// TwinCAT 3 PLC project Untitled1
// ProgramVersion: 3.1.4024.0
// libraries:
//   Tc2_MC2, * (Beckhoff Automation GmbH)
//   Tc2_NCI, * (Beckhoff Automation GmbH)
//   Tc2_Standard, * (Beckhoff Automation GmbH)
//   Tc2_System, * (Beckhoff Automation GmbH)
//   Tc3_Module, * (Beckhoff Automation GmbH)
//   VisuDialogs, * (System)
//   VisuSymbols,3.5.10.0,System
// project tree:
//   DUTs/ MC_CMD.TcDUT, MC_Status.TcDUT
//   / GlobalTextList.TcGTLO, PlcTask.TcTTO, Visualization Manager.TcVMO (not stored)
//   GVLs/ GVL.TcGVL
//   POUs/ MAIN.TcPOU, PANEL.TcPOU, FB_NCI.TcPOU, FB_PowerAll.TcPOU, X_Axis.TcPOU, Y_Axis.TcPOU, Z_Axis.TcPOU
//   VISUs/ Panel.TcVIS

CONFIGURATION Untitled1
    RESOURCE PLC ON TwinCAT3
        TASK PlcTask(INTERVAL := T#10ms, PRIORITY := 20);
        PROGRAM MAIN WITH PlcTask : MAIN;
    END_RESOURCE
END_CONFIGURATION

// ---- DUTs/MC_CMD.TcDUT
TYPE MC_CMD :
STRUCT
	bExe:BOOL;
	lrVelocity:LREAL;
	lrAcceleration:LREAL;
	LrDeceleration:LREAL;
	lrJerk:LREAL;
	lrDistance:LREAL;
	lrPosition:LREAL;
	EnuDirection:  MC_Direction;
	EnuBufferMode: MC_BufferMode;
	EnuOptions  :  ST_MoveOptions;
END_STRUCT
END_TYPE

// ---- DUTs/MC_Status.TcDUT
TYPE MC_Status :
STRUCT
	
	Status   : BOOL;
	Done   : BOOL;
	Busy   : BOOL;
	Error   : BOOL;
	Active   : BOOL;
	CmdAborted   : BOOL;
	InVelocity   : BOOL;
	ErrorID   : UDINT;
	
	
END_STRUCT
END_TYPE

// ---- GVLs/GVL.TcGVL
{attribute 'qualified_only'}
VAR_GLOBAL
	
	BT_Z_AXIS_UP AT %I*:BOOL;
	BT_Z_AXIS_DOWN AT %I*:BOOL;
	SENSOR_Z_AXIS_UP AT %I*:BOOL;
	SENSOR_Z_AXIS_DOWN AT %I*:BOOL;
	Z_AXIS_UP AT %Q*:BOOL;
	Z_AXIS_DOWN AT %Q*:BOOL;
	
	BT_X_AXIS_FRONT AT %I*:BOOL;
	BT_X_AXIS_BACK AT %I*:BOOL;
	BT_Y_AXIS_FRONT AT %I*:BOOL;
	BT_Y_AXIS_BACK AT %I*:BOOL;
	
	X_Position:DINT;
	Y_Position:DINT;
	XY_Velocity: DINT;
	
	X_Current:LREAL;
	Y_Current:LREAL;
	X_Current_INT:DINT;
	Y_Current_INT:DINT;

	Axis_X : AXIS_REF;
	
	X_AxisPower : MC_Power;
	X_AxisReset : MC_Reset;
	X_AxisJog   : MC_Jog;
	X_AxisHome   : MC_Home;
	X_Axis_MovVel1  : MC_MoveVelocity;
	X_Axis_MovVel2  : MC_MoveVelocity;
	X_Axis_MovRel1  : MC_MoveRelative;
	X_Axis_MovRel2  : MC_MoveRelative;
	X_Axis_MovAbs1  : MC_MoveAbsolute;
	X_Axis_MovAbs2  : MC_MoveAbsolute;
	
	X_Axis_Halt     : MC_Halt;
	X_Axis_Stop     : MC_Stop;
	
	X_Read_Pos     : MC_ReadActualPosition;
	Y_Read_Pos     : MC_ReadActualPosition;
	
	// Input command
	X_ResetExe : BOOL;
	
	X_PowerEnable          : BOOL;
	X_PowerEnPositive      : BOOL;
	X_PowerEnNegative      : BOOL;
	
	X_HomeExe              : BOOL;
	X_HomeCamInput 		   : BOOL;
	
	X_JogForward   		   :BOOL;
	X_JogRevise            :BOOL;
	
	X_HaltExe            :BOOL;
	X_StopExe            :BOOL;
	
	X_ST_VelCmd1  : MC_CMD;
	X_ST_VelCmd2  : MC_CMD;
	X_ST_RelCmd1  : MC_CMD;
	X_ST_RelCmd2  : MC_CMD;
	X_ST_AbsCmd1  : MC_CMD;
	X_ST_AbsCmd2  : MC_CMD;
	//
	X_ST_RealPos  :MC_Status;
	Y_ST_RealPos  :MC_Status;
	
	
	X_PowerOverride:  LREAL;
	X_HomePosition:  LREAL;
	X_SetPosition:  LREAL;
	X_JogVelocity:  LREAL;
	
	// Status
	X_ST_Reset           : MC_Status;
	X_ST_Power           : MC_Status;
	X_ST_Home            : MC_Status;
	X_ST_SetPosition     : MC_Status;
	X_ST_Jog             : MC_Status;
	
	X_ST_VelSts1    : MC_Status;
	X_ST_VelSts2    : MC_Status;
	X_ST_RelSts1    : MC_Status;
	X_ST_RelSts2    : MC_Status;
	X_ST_AbsSts1    : MC_Status;
	X_ST_AbsSts2    : MC_Status;
	
	X_ST_Halt          	:MC_Status;
	X_ST_Stop			:MC_Status;
	
	Axis_Y : AXIS_REF;
	
	Y_AxisPower : MC_Power;
	Y_AxisReset : MC_Reset;
	Y_AxisJog   : MC_Jog;
	Y_AxisHome   : MC_Home;
	Y_Axis_MovVel1  : MC_MoveVelocity;
	Y_Axis_MovVel2  : MC_MoveVelocity;
	Y_Axis_MovRel1  : MC_MoveRelative;
	Y_Axis_MovRel2  : MC_MoveRelative;
	Y_Axis_MovAbs1  : MC_MoveAbsolute;
	Y_Axis_MovAbs2  : MC_MoveAbsolute;
	
	Y_Axis_Halt     : MC_Halt;
	Y_Axis_Stop     : MC_Stop;
	
	// Input command
	Y_ResetExe : BOOL;
	
	Y_PowerEnable          : BOOL;
	Y_PowerEnPositive      : BOOL;
	Y_PowerEnNegative      : BOOL;
	
	Y_HomeExe              : BOOL;
	Y_HomeCamInput 		   : BOOL;
	
	Y_JogForward   		   :BOOL;
	Y_JogRevise            :BOOL;
	
	Y_HaltExe            :BOOL;
	Y_StopExe            :BOOL;
	
	Y_ST_VelCmd1  : MC_CMD;
	Y_ST_VelCmd2  : MC_CMD;
	Y_ST_RelCmd1  : MC_CMD;
	Y_ST_RelCmd2  : MC_CMD;
	Y_ST_AbsCmd1  : MC_CMD;
	Y_ST_AbsCmd2  : MC_CMD;
	
	
	Y_PowerOverride:  LREAL;
	Y_HomePosition:  LREAL;
	Y_SetPosition:  LREAL;
	Y_JogVelocity:  LREAL;
	
	// Status
	Y_ST_Reset           : MC_Status;
	Y_ST_Power           : MC_Status;
	Y_ST_Home            : MC_Status;
	Y_ST_SetPosition     : MC_Status;
	Y_ST_Jog             : MC_Status;
	
	Y_ST_VelSts1    : MC_Status;
	Y_ST_VelSts2    : MC_Status;
	Y_ST_RelSts1    : MC_Status;
	Y_ST_RelSts2    : MC_Status;
	Y_ST_AbsSts1    : MC_Status;
	Y_ST_AbsSts2    : MC_Status;
	
	Y_ST_Halt          	:MC_Status;
	Y_ST_Stop			:MC_Status;

	LOAD_PROGRAM : BOOL;
	RUN          : BOOL;
	
END_VAR

// ---- POUs/MAIN.TcPOU
PROGRAM MAIN
VAR
	fbnci :FB_NCI;
	
	stChannelInput  AT %I*: NCTOPLC_NCICHANNEL_REF;
	stChannelOutput AT %Q*: PLCTONC_NCICHANNEL_REF;


END_VAR


X_Axis();
Y_Axis();
Z_Axis();
PANEL();

fbnci(
	sProgramName:='mdi_2.nc' , 
	stChannelInput:=stChannelInput , 
	stChannelOutput:=stChannelOutput , 
	stAxRefAxX:=gvl.Axis_X , 
	stAxRefAyY:=gvl.Axis_Y );

END_PROGRAM

// ---- POUs/FB_NCI.TcPOU
FUNCTION_BLOCK FB_NCI
VAR_INPUT
	sProgramName: STRING;
END_VAR
VAR_IN_OUT
	stChannelInput : NCTOPLC_NCICHANNEL_REF;
	stChannelOutput: PLCTONC_NCICHANNEL_REF;
	
	stAxRefAxX:AXIS_REF;
	stAxRefAyY:AXIS_REF;
END_VAR
VAR
	fbpowerAll   : FB_PowerAll;
	fOverride    :LREAL :=100;
	fbcfgbuildExtgroup : CfgbuildExt3Dgroup;
	fbItpResetEx2      : ItpResetEx2;
	fbItpLoadProgEx    : ItpLoadProgEx;
	fbReconfig         : CfgReconfigGroup;
	fbItpStartStopEx   : ItpStartStopEx;
	
	ItpErrId: UDINT;
	ItpState: UDINT;
	ItpStateErr: BOOL;
	ItpStateIdle: BOOL;
	ItpStateReady: BOOL;
	ItpStateRunning: BOOL;
	ItpStateAborted: BOOL;
END_VAR



fbpowerAll(
	bEnable:=GVL.X_PowerEnable , 
	bStatus=> , 
	bError=> , 
	stAxRefAxX:= stAxRefAxX, 
	stAxRefAyY:= stAxRefAyY);
	
	ItpSetOverridePercent(fOverridePercent:= fOverride, sPlcToNci:=stChannelOutput);
fbcfgbuildExtgroup(
	bExecute:= GVL.X_PowerEnable, //fbcfgbuildExtgroup.bExecute, 
	nGroupId:= stChannelInput.GrpId, 
	nXAxisId:= stAxRefAxX.NcToPlc.AxisId, 
	nYAxisId:= stAxRefAyY.NcToPlc.AxisId,
	nZAxisId:= , 
	nQ1AxisId:= , 
	nQ2AxisId:= , 
	nQ3AxisId:= , 
	nQ4AxisId:= , 
	nQ5AxisId:= , 
	tTimeOut:= fbcfgbuildExtgroup.tTimeOut, 
	bBusy=> , 
	bErr=> , 
	nErrId=> );
	
fbItpResetEx2(
	bExecute:= fbItpResetEx2.bExecute, 
	tTimeOut:= fbItpResetEx2.tTimeOut, 
	sNciToPlc:= stChannelInput, 
	bBusy=> , 
	bErr=> , 
	nErrId=> );
	
fbItpLoadProgEx(
	sNciToPlc:= stChannelInput , 
	bExecute:= GVL.LOAD_PROGRAM,//fbItpLoadProgEx.bExecute, 
	sPrg:= sProgramName, 
	nLength:= LEN(sProgramName), 
	tTimeOut:= fbItpLoadProgEx.tTimeOut, 
	bBusy=> , 
	bErr=> , 
	nErrId=> );
	
	ItpState := stChannelInput.ItpState;
	ItpStateReady := ItpState = NCI_INTERPRETER_READY;
	
fbItpStartStopEx(
	bStart:=GVL.RUN,//fbItpStartStopEx.bStart , 
	bStop:= fbItpStartStopEx.bStop, 
	tTimeOut:=fbItpStartStopEx.tTimeout , 
	sNciToPlc:= stChannelInput, 
	bBusy=> , 
	bErr=> , 
	nErrId=> );

fbReconfig(
	bExecute:=fbReconfig.bExecute , 
	nGroupId:= stChannelInput.GrpId, 
	tTimeOut:= , 
	bBusy=> , 
	bErr=> , 
	nErrId=> );

END_FUNCTION_BLOCK

// ---- POUs/FB_PowerAll.TcPOU
FUNCTION_BLOCK FB_PowerAll
VAR_INPUT
	bEnable: BOOL;
END_VAR
VAR_OUTPUT
	bStatus:BOOL;
	bError :BOOL;
END_VAR
VAR_IN_OUT
	stAxRefAxX:AXIS_REF;
	stAxRefAyY:AXIS_REF;	
END_VAR
VAR
	fbPower1:MC_Power;
	fbPower2:MC_Power;
	
END_VAR

// power all axis//
fbPower1(
	Axis:=stAxRefAxX , 
	Enable:=bEnable , 
	Enable_Positive:= TRUE, 
	Enable_Negative:=TRUE , 
	Override:=100 , 
	BufferMode:= , 
	Options:= , 
	Status=> , 
	Busy=> , 
	Error=> , 
	ErrorID=> );
	
fbPower2(
	Axis:=stAxRefAyY , 
	Enable:=bEnable , 
	Enable_Positive:= TRUE, 
	Enable_Negative:=TRUE , 
	Override:=100 , 
	BufferMode:= , 
	Options:= , 
	Status=> , 
	Busy=> , 
	Error=> , 
	ErrorID=> );
	
	
bStatus :=fbPower1.Status AND fbPower2.Status;
bError  :=fbPower1.Status OR  fbPower2.Status;

END_FUNCTION_BLOCK

// ---- POUs/X_Axis.TcPOU
PROGRAM X_Axis
VAR

END_VAR



TrucX();

METHOD nhap : BOOL
VAR_INPUT
END_VAR
// NETWORK 1

// NETWORK 2
END_METHOD

METHOD TrucX : BOOL
VAR_INPUT
END_VAR
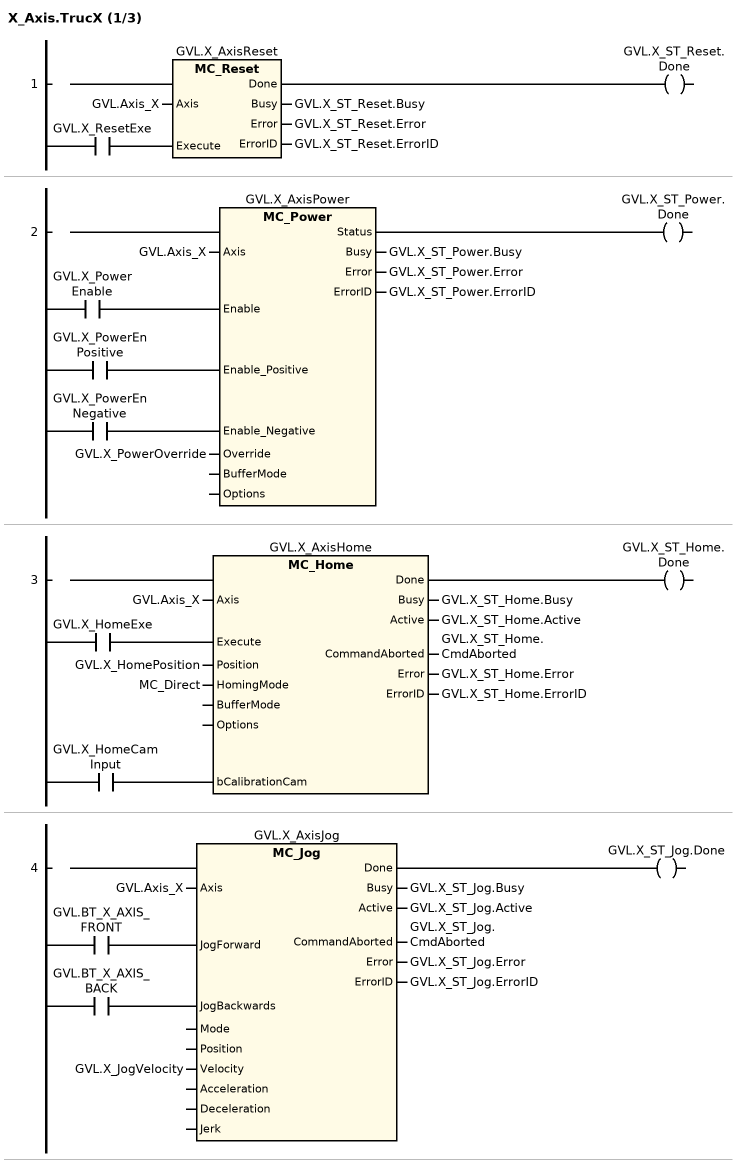
// NETWORK 1
GVL.X_AxisReset(
    Axis := GVL.Axis_X,
    Execute := GVL.X_ResetExe,
    Busy => GVL.X_ST_Reset.Busy,
    Error => GVL.X_ST_Reset.Error,
    ErrorID => GVL.X_ST_Reset.ErrorID); // MC_Reset
GVL.X_ST_Reset.Done := GVL.X_AxisReset.Done;

// NETWORK 2
GVL.X_AxisPower(
    Axis := GVL.Axis_X,
    Enable := GVL.X_PowerEnable,
    Enable_Positive := GVL.X_PowerEnPositive,
    Enable_Negative := GVL.X_PowerEnNegative,
    Override := GVL.X_PowerOverride,
    Busy => GVL.X_ST_Power.Busy,
    Error => GVL.X_ST_Power.Error,
    ErrorID => GVL.X_ST_Power.ErrorID); // MC_Power
GVL.X_ST_Power.Done := GVL.X_AxisPower.Status;

// NETWORK 3
GVL.X_AxisHome(
    Axis := GVL.Axis_X,
    Execute := GVL.X_HomeExe,
    Position := GVL.X_HomePosition,
    HomingMode := MC_Direct,
    bCalibrationCam := GVL.X_HomeCamInput,
    Busy => GVL.X_ST_Home.Busy,
    Active => GVL.X_ST_Home.Active,
    CommandAborted => GVL.X_ST_Home.CmdAborted,
    Error => GVL.X_ST_Home.Error,
    ErrorID => GVL.X_ST_Home.ErrorID); // MC_Home
GVL.X_ST_Home.Done := GVL.X_AxisHome.Done;

// NETWORK 4
GVL.X_AxisJog(
    Axis := GVL.Axis_X,
    JogForward := GVL.BT_X_AXIS_FRONT,
    JogBackwards := GVL.BT_X_AXIS_BACK,
    Velocity := GVL.X_JogVelocity,
    Busy => GVL.X_ST_Jog.Busy,
    Active => GVL.X_ST_Jog.Active,
    CommandAborted => GVL.X_ST_Jog.CmdAborted,
    Error => GVL.X_ST_Jog.Error,
    ErrorID => GVL.X_ST_Jog.ErrorID); // MC_Jog
GVL.X_ST_Jog.Done := GVL.X_AxisJog.Done;

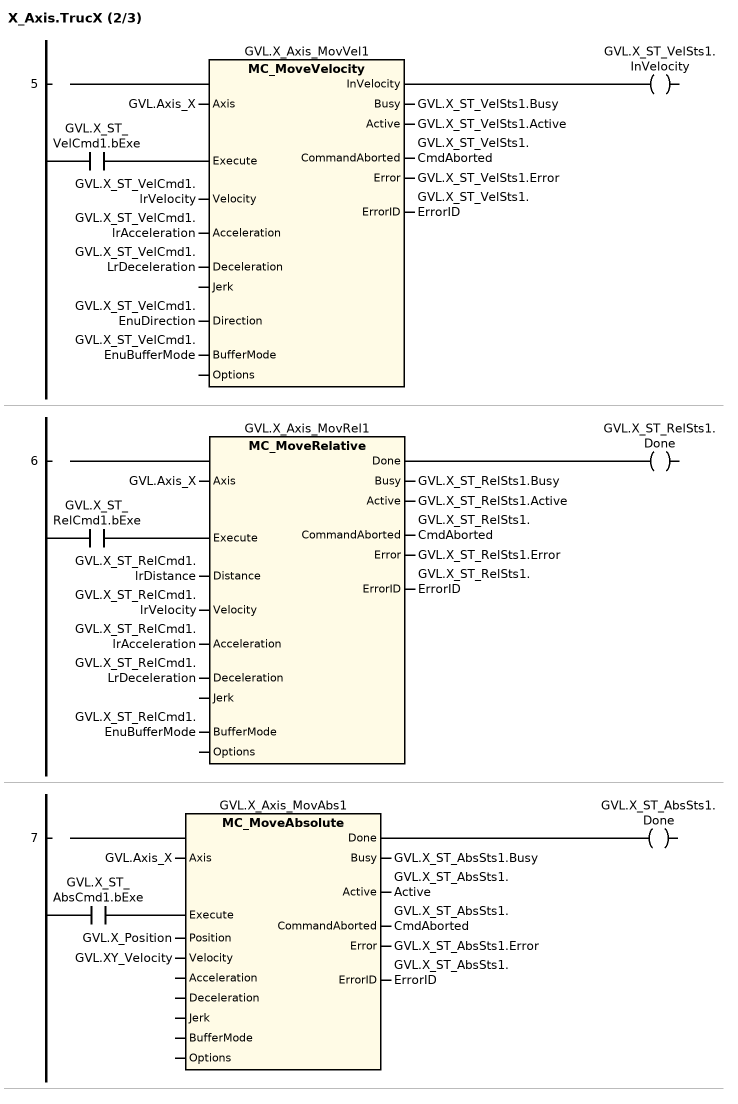
// NETWORK 5
GVL.X_Axis_MovVel1(
    Axis := GVL.Axis_X,
    Execute := GVL.X_ST_VelCmd1.bExe,
    Velocity := GVL.X_ST_VelCmd1.lrVelocity,
    Acceleration := GVL.X_ST_VelCmd1.lrAcceleration,
    Deceleration := GVL.X_ST_VelCmd1.LrDeceleration,
    Direction := GVL.X_ST_VelCmd1.EnuDirection,
    BufferMode := GVL.X_ST_VelCmd1.EnuBufferMode,
    Busy => GVL.X_ST_VelSts1.Busy,
    Active => GVL.X_ST_VelSts1.Active,
    CommandAborted => GVL.X_ST_VelSts1.CmdAborted,
    Error => GVL.X_ST_VelSts1.Error,
    ErrorID => GVL.X_ST_VelSts1.ErrorID); // MC_MoveVelocity
GVL.X_ST_VelSts1.InVelocity := GVL.X_Axis_MovVel1.InVelocity;

// NETWORK 6
GVL.X_Axis_MovRel1(
    Axis := GVL.Axis_X,
    Execute := GVL.X_ST_RelCmd1.bExe,
    Distance := GVL.X_ST_RelCmd1.lrDistance,
    Velocity := GVL.X_ST_RelCmd1.lrVelocity,
    Acceleration := GVL.X_ST_RelCmd1.lrAcceleration,
    Deceleration := GVL.X_ST_RelCmd1.LrDeceleration,
    BufferMode := GVL.X_ST_RelCmd1.EnuBufferMode,
    Busy => GVL.X_ST_RelSts1.Busy,
    Active => GVL.X_ST_RelSts1.Active,
    CommandAborted => GVL.X_ST_RelSts1.CmdAborted,
    Error => GVL.X_ST_RelSts1.Error,
    ErrorID => GVL.X_ST_RelSts1.ErrorID); // MC_MoveRelative
GVL.X_ST_RelSts1.Done := GVL.X_Axis_MovRel1.Done;

// NETWORK 7
GVL.X_Axis_MovAbs1(
    Axis := GVL.Axis_X,
    Execute := GVL.X_ST_AbsCmd1.bExe,
    Position := GVL.X_Position,
    Velocity := GVL.XY_Velocity,
    Busy => GVL.X_ST_AbsSts1.Busy,
    Active => GVL.X_ST_AbsSts1.Active,
    CommandAborted => GVL.X_ST_AbsSts1.CmdAborted,
    Error => GVL.X_ST_AbsSts1.Error,
    ErrorID => GVL.X_ST_AbsSts1.ErrorID); // MC_MoveAbsolute
GVL.X_ST_AbsSts1.Done := GVL.X_Axis_MovAbs1.Done;

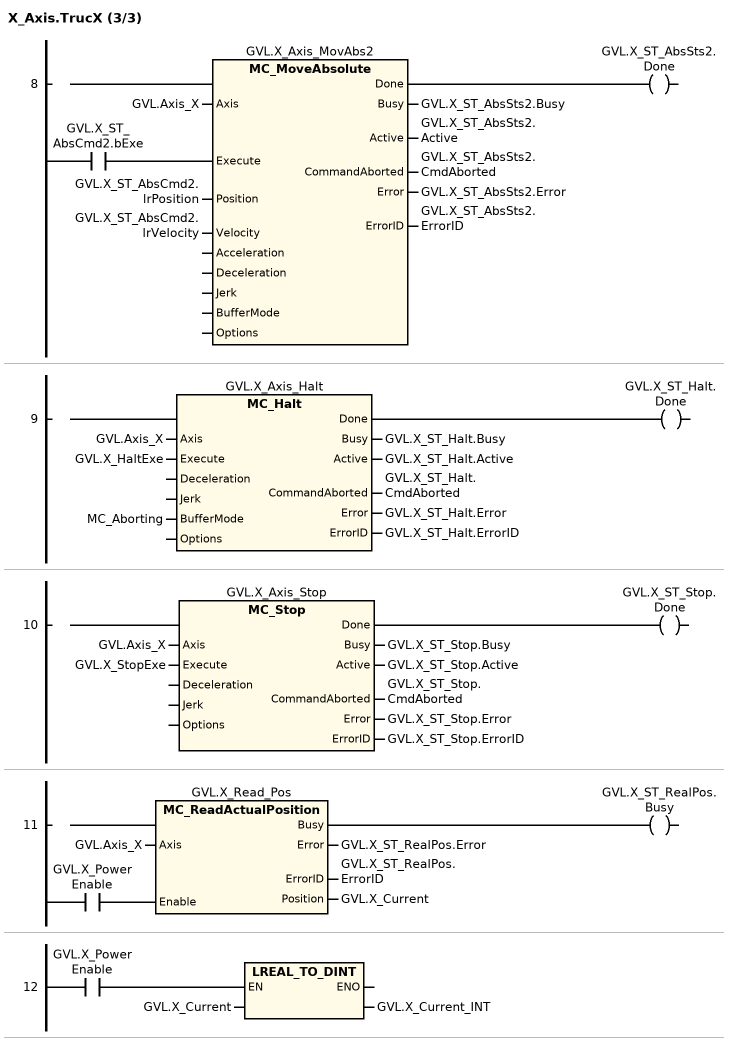
// NETWORK 8
GVL.X_Axis_MovAbs2(
    Axis := GVL.Axis_X,
    Execute := GVL.X_ST_AbsCmd2.bExe,
    Position := GVL.X_ST_AbsCmd2.lrPosition,
    Velocity := GVL.X_ST_AbsCmd2.lrVelocity,
    Busy => GVL.X_ST_AbsSts2.Busy,
    Active => GVL.X_ST_AbsSts2.Active,
    CommandAborted => GVL.X_ST_AbsSts2.CmdAborted,
    Error => GVL.X_ST_AbsSts2.Error,
    ErrorID => GVL.X_ST_AbsSts2.ErrorID); // MC_MoveAbsolute
GVL.X_ST_AbsSts2.Done := GVL.X_Axis_MovAbs2.Done;

// NETWORK 9
GVL.X_Axis_Halt(
    Axis := GVL.Axis_X,
    Execute := GVL.X_HaltExe,
    BufferMode := MC_Aborting,
    Busy => GVL.X_ST_Halt.Busy,
    Active => GVL.X_ST_Halt.Active,
    CommandAborted => GVL.X_ST_Halt.CmdAborted,
    Error => GVL.X_ST_Halt.Error,
    ErrorID => GVL.X_ST_Halt.ErrorID); // MC_Halt
GVL.X_ST_Halt.Done := GVL.X_Axis_Halt.Done;

// NETWORK 10
GVL.X_Axis_Stop(
    Axis := GVL.Axis_X,
    Execute := GVL.X_StopExe,
    Busy => GVL.X_ST_Stop.Busy,
    Active => GVL.X_ST_Stop.Active,
    CommandAborted => GVL.X_ST_Stop.CmdAborted,
    Error => GVL.X_ST_Stop.Error,
    ErrorID => GVL.X_ST_Stop.ErrorID); // MC_Stop
GVL.X_ST_Stop.Done := GVL.X_Axis_Stop.Done;

// NETWORK 11
GVL.X_Read_Pos(
    Axis := GVL.Axis_X,
    Enable := GVL.X_PowerEnable,
    Busy => GVL.X_ST_RealPos.Busy,
    Error => GVL.X_ST_RealPos.Error,
    ErrorID => GVL.X_ST_RealPos.ErrorID,
    Position => GVL.X_Current); // MC_ReadActualPosition

// NETWORK 12
IF GVL.X_PowerEnable THEN GVL.X_Current_INT := LREAL_TO_DINT(GVL.X_Current); END_IF
END_METHOD

END_PROGRAM

// ---- POUs/Y_Axis.TcPOU
PROGRAM Y_Axis
VAR

END_VAR



TrucY();

METHOD TrucY : BOOL
VAR_INPUT
END_VAR
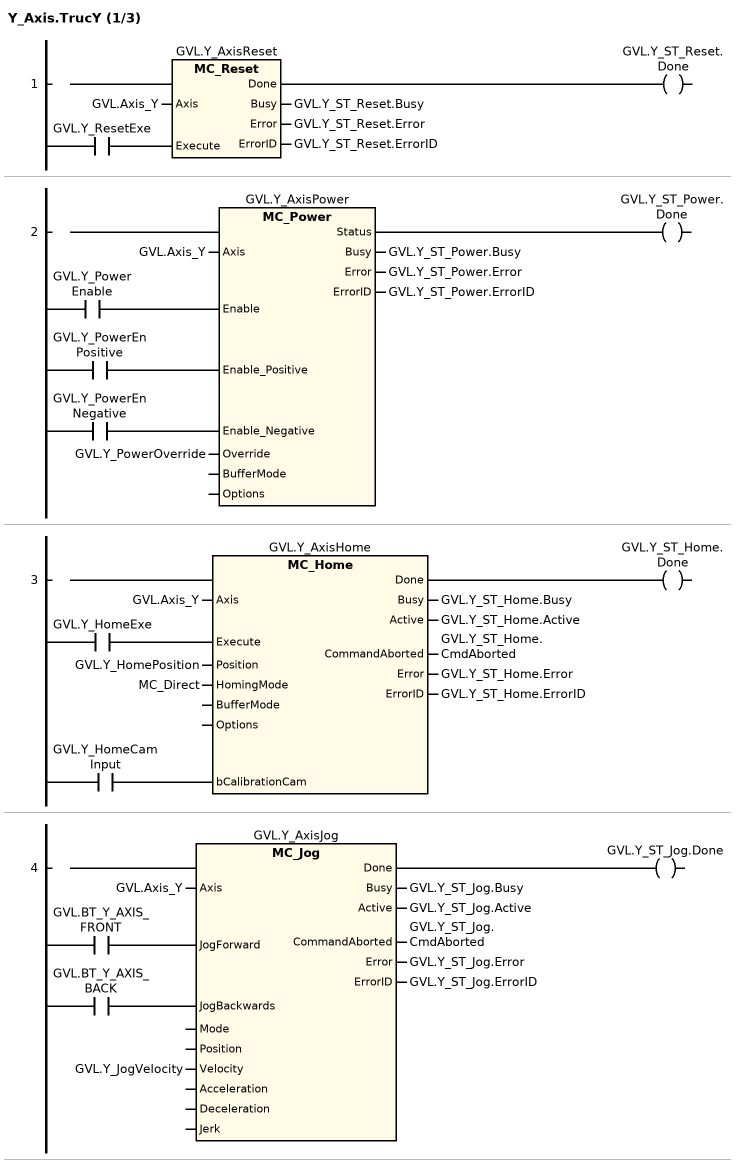
// NETWORK 1
GVL.Y_AxisReset(
    Axis := GVL.Axis_Y,
    Execute := GVL.Y_ResetExe,
    Busy => GVL.Y_ST_Reset.Busy,
    Error => GVL.Y_ST_Reset.Error,
    ErrorID => GVL.Y_ST_Reset.ErrorID); // MC_Reset
GVL.Y_ST_Reset.Done := GVL.Y_AxisReset.Done;

// NETWORK 2
GVL.Y_AxisPower(
    Axis := GVL.Axis_Y,
    Enable := GVL.Y_PowerEnable,
    Enable_Positive := GVL.Y_PowerEnPositive,
    Enable_Negative := GVL.Y_PowerEnNegative,
    Override := GVL.Y_PowerOverride,
    Busy => GVL.Y_ST_Power.Busy,
    Error => GVL.Y_ST_Power.Error,
    ErrorID => GVL.Y_ST_Power.ErrorID); // MC_Power
GVL.Y_ST_Power.Done := GVL.Y_AxisPower.Status;

// NETWORK 3
GVL.Y_AxisHome(
    Axis := GVL.Axis_Y,
    Execute := GVL.Y_HomeExe,
    Position := GVL.Y_HomePosition,
    HomingMode := MC_Direct,
    bCalibrationCam := GVL.Y_HomeCamInput,
    Busy => GVL.Y_ST_Home.Busy,
    Active => GVL.Y_ST_Home.Active,
    CommandAborted => GVL.Y_ST_Home.CmdAborted,
    Error => GVL.Y_ST_Home.Error,
    ErrorID => GVL.Y_ST_Home.ErrorID); // MC_Home
GVL.Y_ST_Home.Done := GVL.Y_AxisHome.Done;

// NETWORK 4
GVL.Y_AxisJog(
    Axis := GVL.Axis_Y,
    JogForward := GVL.BT_Y_AXIS_FRONT,
    JogBackwards := GVL.BT_Y_AXIS_BACK,
    Velocity := GVL.Y_JogVelocity,
    Busy => GVL.Y_ST_Jog.Busy,
    Active => GVL.Y_ST_Jog.Active,
    CommandAborted => GVL.Y_ST_Jog.CmdAborted,
    Error => GVL.Y_ST_Jog.Error,
    ErrorID => GVL.Y_ST_Jog.ErrorID); // MC_Jog
GVL.Y_ST_Jog.Done := GVL.Y_AxisJog.Done;

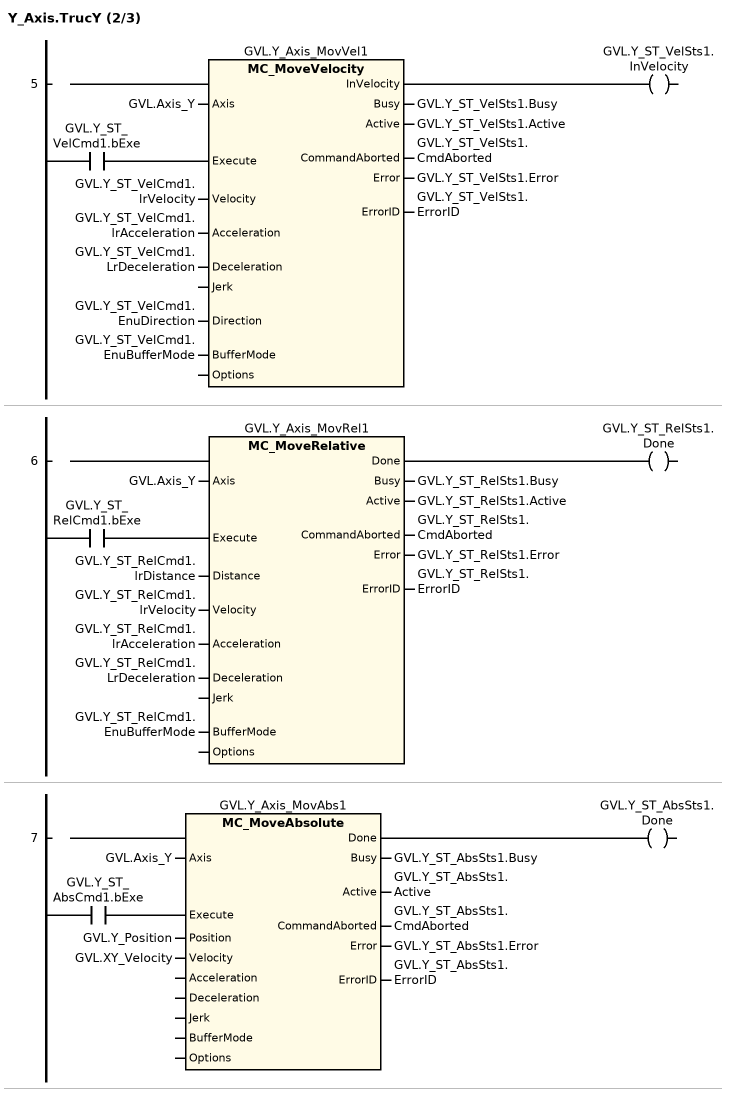
// NETWORK 5
GVL.Y_Axis_MovVel1(
    Axis := GVL.Axis_Y,
    Execute := GVL.Y_ST_VelCmd1.bExe,
    Velocity := GVL.Y_ST_VelCmd1.lrVelocity,
    Acceleration := GVL.Y_ST_VelCmd1.lrAcceleration,
    Deceleration := GVL.Y_ST_VelCmd1.LrDeceleration,
    Direction := GVL.Y_ST_VelCmd1.EnuDirection,
    BufferMode := GVL.Y_ST_VelCmd1.EnuBufferMode,
    Busy => GVL.Y_ST_VelSts1.Busy,
    Active => GVL.Y_ST_VelSts1.Active,
    CommandAborted => GVL.Y_ST_VelSts1.CmdAborted,
    Error => GVL.Y_ST_VelSts1.Error,
    ErrorID => GVL.Y_ST_VelSts1.ErrorID); // MC_MoveVelocity
GVL.Y_ST_VelSts1.InVelocity := GVL.Y_Axis_MovVel1.InVelocity;

// NETWORK 6
GVL.Y_Axis_MovRel1(
    Axis := GVL.Axis_Y,
    Execute := GVL.Y_ST_RelCmd1.bExe,
    Distance := GVL.Y_ST_RelCmd1.lrDistance,
    Velocity := GVL.Y_ST_RelCmd1.lrVelocity,
    Acceleration := GVL.Y_ST_RelCmd1.lrAcceleration,
    Deceleration := GVL.Y_ST_RelCmd1.LrDeceleration,
    BufferMode := GVL.Y_ST_RelCmd1.EnuBufferMode,
    Busy => GVL.Y_ST_RelSts1.Busy,
    Active => GVL.Y_ST_RelSts1.Active,
    CommandAborted => GVL.Y_ST_RelSts1.CmdAborted,
    Error => GVL.Y_ST_RelSts1.Error,
    ErrorID => GVL.Y_ST_RelSts1.ErrorID); // MC_MoveRelative
GVL.Y_ST_RelSts1.Done := GVL.Y_Axis_MovRel1.Done;

// NETWORK 7
GVL.Y_Axis_MovAbs1(
    Axis := GVL.Axis_Y,
    Execute := GVL.Y_ST_AbsCmd1.bExe,
    Position := GVL.Y_Position,
    Velocity := GVL.XY_Velocity,
    Busy => GVL.Y_ST_AbsSts1.Busy,
    Active => GVL.Y_ST_AbsSts1.Active,
    CommandAborted => GVL.Y_ST_AbsSts1.CmdAborted,
    Error => GVL.Y_ST_AbsSts1.Error,
    ErrorID => GVL.Y_ST_AbsSts1.ErrorID); // MC_MoveAbsolute
GVL.Y_ST_AbsSts1.Done := GVL.Y_Axis_MovAbs1.Done;

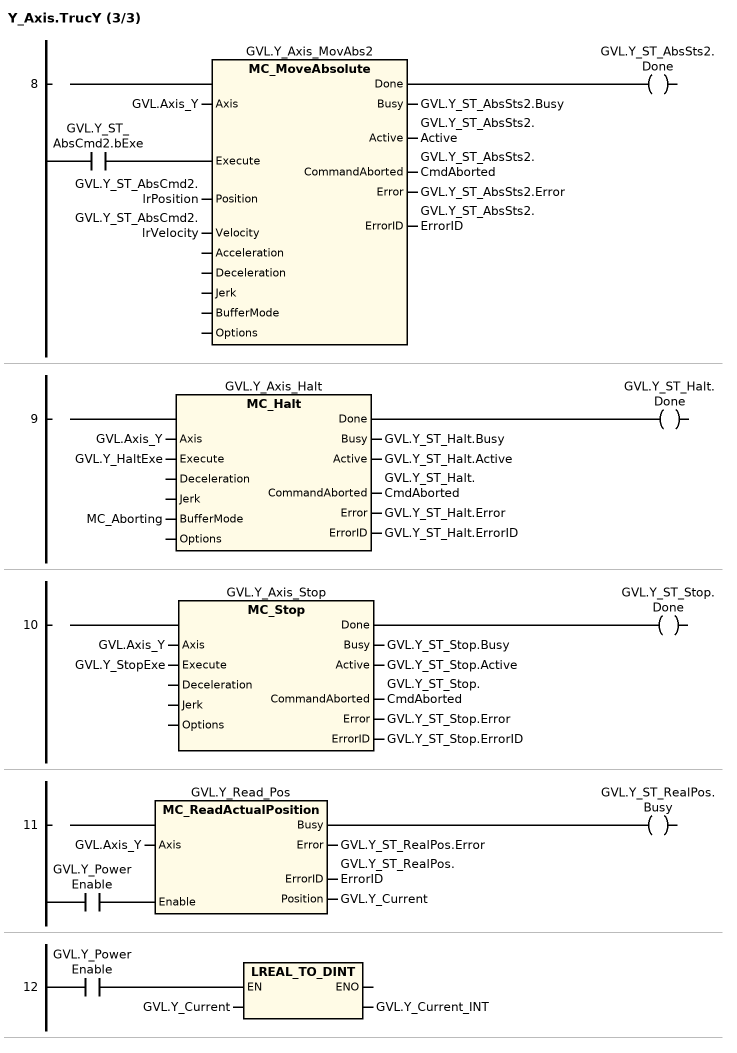
// NETWORK 8
GVL.Y_Axis_MovAbs2(
    Axis := GVL.Axis_Y,
    Execute := GVL.Y_ST_AbsCmd2.bExe,
    Position := GVL.Y_ST_AbsCmd2.lrPosition,
    Velocity := GVL.Y_ST_AbsCmd2.lrVelocity,
    Busy => GVL.Y_ST_AbsSts2.Busy,
    Active => GVL.Y_ST_AbsSts2.Active,
    CommandAborted => GVL.Y_ST_AbsSts2.CmdAborted,
    Error => GVL.Y_ST_AbsSts2.Error,
    ErrorID => GVL.Y_ST_AbsSts2.ErrorID); // MC_MoveAbsolute
GVL.Y_ST_AbsSts2.Done := GVL.Y_Axis_MovAbs2.Done;

// NETWORK 9
GVL.Y_Axis_Halt(
    Axis := GVL.Axis_Y,
    Execute := GVL.Y_HaltExe,
    BufferMode := MC_Aborting,
    Busy => GVL.Y_ST_Halt.Busy,
    Active => GVL.Y_ST_Halt.Active,
    CommandAborted => GVL.Y_ST_Halt.CmdAborted,
    Error => GVL.Y_ST_Halt.Error,
    ErrorID => GVL.Y_ST_Halt.ErrorID); // MC_Halt
GVL.Y_ST_Halt.Done := GVL.Y_Axis_Halt.Done;

// NETWORK 10
GVL.Y_Axis_Stop(
    Axis := GVL.Axis_Y,
    Execute := GVL.Y_StopExe,
    Busy => GVL.Y_ST_Stop.Busy,
    Active => GVL.Y_ST_Stop.Active,
    CommandAborted => GVL.Y_ST_Stop.CmdAborted,
    Error => GVL.Y_ST_Stop.Error,
    ErrorID => GVL.Y_ST_Stop.ErrorID); // MC_Stop
GVL.Y_ST_Stop.Done := GVL.Y_Axis_Stop.Done;

// NETWORK 11
GVL.Y_Read_Pos(
    Axis := GVL.Axis_Y,
    Enable := GVL.Y_PowerEnable,
    Busy => GVL.Y_ST_RealPos.Busy,
    Error => GVL.Y_ST_RealPos.Error,
    ErrorID => GVL.Y_ST_RealPos.ErrorID,
    Position => GVL.Y_Current); // MC_ReadActualPosition

// NETWORK 12
IF GVL.Y_PowerEnable THEN GVL.Y_Current_INT := LREAL_TO_DINT(GVL.Y_Current); END_IF
END_METHOD

END_PROGRAM

// ---- POUs/Z_Axis.TcPOU
PROGRAM Z_Axis
VAR
	HMI_Z_UP : BOOL;
	HMI_Z_DOWN : BOOL;
END_VAR

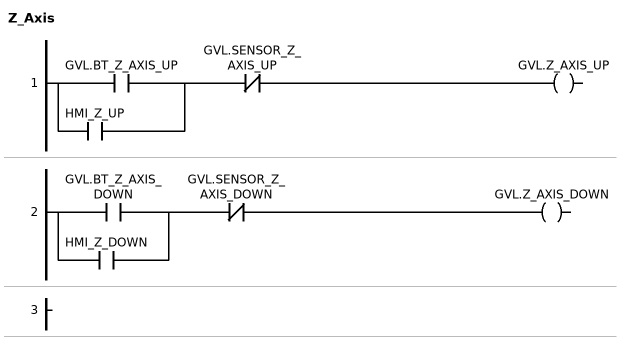
// NETWORK 1
GVL.Z_AXIS_UP := (GVL.BT_Z_AXIS_UP OR HMI_Z_UP) AND NOT GVL.SENSOR_Z_AXIS_UP;

// NETWORK 2
GVL.Z_AXIS_DOWN := (GVL.BT_Z_AXIS_DOWN OR HMI_Z_DOWN) AND NOT GVL.SENSOR_Z_AXIS_DOWN;

// NETWORK 3

END_PROGRAM

// ---- POUs/PANEL.TcPOU
PROGRAM PANEL
VAR
	START:BOOL;
	STOP:BOOL;
	HOME:BOOL;
	WRITE:BOOL;
	M00:BOOL;
	M01:BOOL;
	TON_0: TON;
	
	
END_VAR
VAR // added by the converter: edge detectors and wires of the graphical bodies
    _w1, _w2, _w3, _w4, _w5 : BOOL;
END_VAR

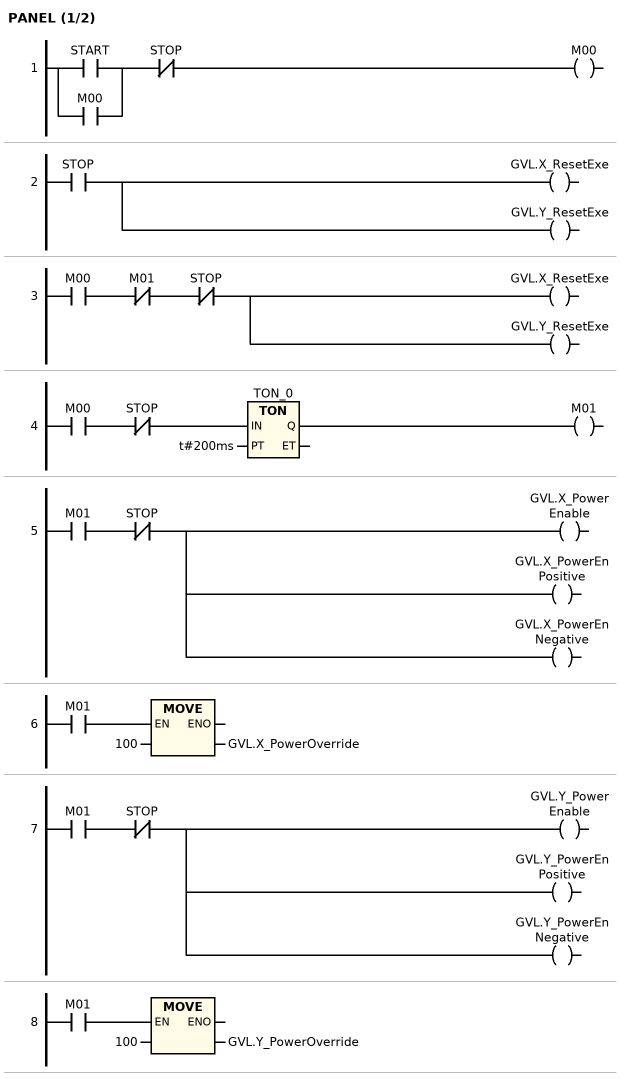
// NETWORK 1
M00 := (START OR M00) AND NOT STOP;

// NETWORK 2
GVL.X_ResetExe := STOP;
GVL.Y_ResetExe := STOP;

// NETWORK 3
_w1 := M00 AND NOT M01 AND NOT STOP;
GVL.X_ResetExe := _w1;
GVL.Y_ResetExe := _w1;

// NETWORK 4
TON_0(IN := M00 AND NOT STOP, PT := t#200ms); // TON
M01 := TON_0.Q;

// NETWORK 5
_w2 := M01 AND NOT STOP;
GVL.X_PowerEnable := _w2;
GVL.X_PowerEnPositive := _w2;
GVL.X_PowerEnNegative := _w2;

// NETWORK 6
IF M01 THEN GVL.X_PowerOverride := 100; END_IF

// NETWORK 7
_w3 := M01 AND NOT STOP;
GVL.Y_PowerEnable := _w3;
GVL.Y_PowerEnPositive := _w3;
GVL.Y_PowerEnNegative := _w3;

// NETWORK 8
IF M01 THEN GVL.Y_PowerOverride := 100; END_IF

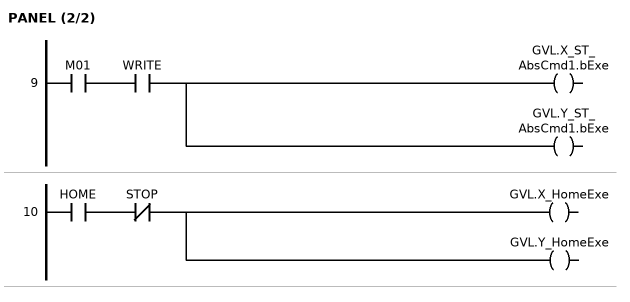
// NETWORK 9
_w4 := M01 AND WRITE;
GVL.X_ST_AbsCmd1.bExe := _w4;
GVL.Y_ST_AbsCmd1.bExe := _w4;

// NETWORK 10
_w5 := HOME AND NOT STOP;
GVL.X_HomeExe := _w5;
GVL.Y_HomeExe := _w5;

END_PROGRAM

// ---- GlobalTextList.TcGTLO
TEXTLIST GlobalTextList
  713 = '15'
  182 = 'X+'
  95 = 'X-'
  539 = 'Y'
  45 = 'Y+'
  157 = 'Y-'
  452 = 'Z+'
  80 = 'Z-'
END_TEXTLIST

// ---- VISUs/Panel.TcVIS
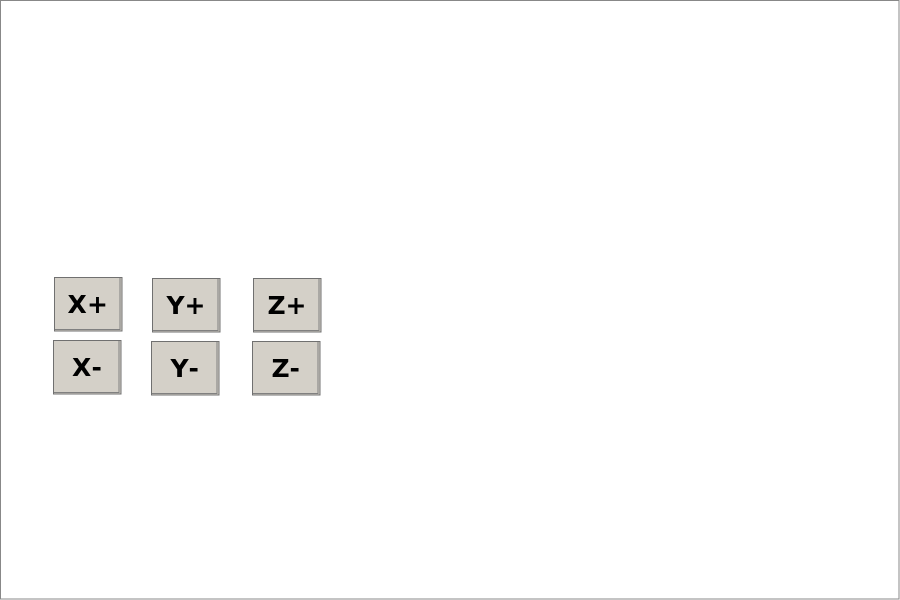
VISUALIZATION Panel  // 900x600
    Button (53,340 68x54), "X-"
        tap GVL.BT_X_AXIS_LEFT
    Button (54,277 68x54), "X+"
        tap GVL.BT_X_AXIS_RIGHT
    Button (152,278 68x54), "Y+"
        tap GVL.BT_Y_AXIS_FRONT
    Button (151,341 68x54), "Y-"
        tap GVL.BT_Y_AXIS_BACK
    Button (253,278 68x54), "Z+"
        tap GVL.Z_AXIS_UP
    Button (252,341 68x54), "Z-"
        tap GVL.Z_AXIS_DOWN
END_VISUALIZATION
